Fanuc KAREL source: kt00070.KL

-- PROVISIONAL review KL for V770-1; original PC SHA256 6577c6c464ec249d208dd1b7b9bf93a80b8b1f9defab26b8e821d05f9fb8ddb3
-- Incomplete behavior may be omitted. Consult companion uncertainty JSON. Do not deploy.
PROGRAM KT00070
%NOLOCKGROUP
VAR
  I1 : INTEGER
  OUT : REAL
-- UNRESOLVED_DECL Y2 type=002018
BEGIN
  -- UNRESOLVED_PC offsets 5-16; opcodes 2E,23
  -- UNRESOLVED_PC offsets 21-35; opcodes 2E,22,9D,33,B2
  -- UNRESOLVED_PC offsets 40-63; opcodes 21,22,9D,33,B1,54,64,23
  -- UNRESOLVED_PC offsets 68-72; opcodes 7F
END KT00070
